# EPICS substitutions: epics/m-epics-eemcu/eemcuApp/Db/Sim8-extra-m3.substitutions
file "eemcu-extra.template"
{
pattern
{P,      M,    R,   PORT, ADDR, PREC, HOMEPROC}
{IOC:,   m3, m3-,   MCU1,    3, 3,    3}
}
